// TIA Portal V16 export
// export: Created 2023-03-29T11:03:26.1112429Z, ExportSetting WithDefaults, DisplayName Totally Integrated Automation Portal, DisplayVersion V16 Update 6, DisplayName TIA Portal Version Control Interface, DisplayVersion V16 Update 2, DisplayName TIA Portal Openness, DisplayVersion V16 Update 6, DisplayName STEP 7 Professional, DisplayVersion V16 Update 6, DisplayName STEP 7 Safety, DisplayVersion V16, DisplayName WinCC Advanced, DisplayVersion V16 Update 6
DATA_BLOCK "dbHoldRegSlave_to_MT101"   // DB100
{ S7_Optimized_Access := 'FALSE' }
VERSION : 0.1
// stored: AutoNumber false, DBAccessibleFromOPCUA true, IsOnlyStoredInLoadMemory false, IsWriteProtectedInAS false
   VAR
      Status_Sterowanie : Struct
         instvValveZ1 : Word := 33924;   // Zasuwa Status Z1
         instvValveZ2 : Word := 33924;   // Zasuwa Status Z2
         instvValveZ3 : Word := 33924;   // Zasuwa Status Z3
         instvValveZ4 : Word := 33924;   // Zasuwa Status Z4
         instvValveZ5 : Word := 33924;   // Zasuwa Status Z5
         instvValveZ6 : Word := 33924;   // Zasuwa Status Z6
         instvValveZ7 : Word := 33924;   // Zasuwa Status Z7
         instvValveZ8 : Word := 33924;   // Zasuwa Status Z8
         instvValveZ9 : Word := 33924;   // Zasuwa Status Z9
         instvValveZ10 : Word := 33924;   // Zasuwa Status Z10
         instControllDrivers_1 : Int;   // Bity sterowania napędami (start, stop, otwórz, zamknij) / Bity sterowania napędami (start, stop, otwórz, zamknij) Pompami M1-M4, Zasuwami Z1, Z2, Z3, Z4
         instControllDrivers_2 : Int;   // Bity przełączenia trybu pracy napędów / Bity sterowania napędami ( otwórz, zamknij, start, stop) Zasuwami Z5, Z6, Z7, Z8, Z9, Z10, Z11, Z12
         instConrol_ManAut_1 : Int;   // Bity przełączenia trybu pracy napędów / Bity przełączenia trybu pracy napędów M1-M4, Zasuwami Z1, Z2, Z3, Z4
         instConrol_ManAut_2 : Int;   // Bity przełączenia trybu pracy napędów / Bity przełączenia trybu pracy napędów Z5, Z6, Z7, Z8, Z9, Z10, Z11, Z12
         instLevelTank1 : Int;   // Poziom zbiornik
         instLevelTank2 : Int;   // Poziom zbiornik
         instLevelTank3 : Int;   // Poziom zbiornik
         instLevelTank4 : Int;   // Poziom zbiornik
         instPosition_Z10 : Real;   // rezerwa / Zadawanie położenia Z10
         instClearFault1 : Int;   // Bity kasowania alarmów napędów M1-M4, Z1 - Z12
         instSygSter_1 : Int;   // rezerwa / Sygnały sterowania strategią pompownia - 0= wyłaczone, 1=dosilanie, 2=przetłaczanie,3=automat, 4=ręczne
         instSygSter_2 : Int;   // Sygnały sterowania cyklem zbiorniki 0-wyłączone, 1=dobowy, 2=tygodniowy, 3=ręczne
         instCurrent_Inverter : Int;   // Aktualny prądu falownika
         instHz_Inverter : Int;   // Aktualne Hz na falowniku
      END_STRUCT;
      Pomiary : Struct
         instLevelSetFilling : Real;   // Zadany poziom napełniania
         instLevelSetEmptying : Real;   // Zadany poziom opróżniania
         instSetbarDN225_B6 : Real;   // Zadany ciśnienie tłóczenia kierunek miasto, Modbus 40035
         instSetbarDN500_B5 : Real;   // Zadana ciśnienie dosilania kierunek dosilanie "0" Modbus 40037
         instSetBarMinB9 : Real;   // Zadawana dolna granica ciśnienia studnia "Granica" Modbus 40039
         instB5bar_act : Real;   // Aktualne ciśnienie zasilania z sieci
         instPozitionZ10_act : Real;   // Aktualna pozycja zasuwy Z10
         instFlowDN500_act : Real;   // Przepływ DN500 (l/s) aktualny, zasilanie zbiorników, DOSILANIE, Modbus 40055
         instFlowDN500_sum : Real;   // SUMA przepływu Dolna DN500 Modbus 40057
      END_STRUCT;
      Godziny : Struct
         instHourStart_Filling : Int;   // Godzina start napełniania
         instMinutStart_Filling : Int;   // Minuta start napełniania
         instHourStop_Filling : Int;   // Godzina stop napełniania
         instMinutStopt_Filling : Int;   // Minuta stop napełniania
         instHourStart_City : Int;   // Godzina start przetłaczanie miasto DN225
         instMinutStart_City : Int;   // Minuty start przetłaczanie miasto DN225
         instHourStop_City : Int;   // Godzina stop przetłaczanie miasto DN225
         instMinutStopt_City : Int;   // Minuty stop przetłaczanie miasto DN225
         instHourStart_Replen : Int;   // Godzina start przetłaczanie magistrala DN500
         instMinutStart_Replen : Int;   // Minuty start przetłaczanie magistrala DN500
         instHourStop_Replen : Int;   // Godzina stop przetłaczanie magistrala DN500
         instMinutStopt_Replen : Int;   // Minuty stop przetłaczanie magistrala DN500
      END_STRUCT;
   END_VAR
BEGIN
END_DATA_BLOCK
